SUBAPPLICATION mapping_Uebung_033_VV_FORTE_PC_B (* LED Strip Blinkende LED *)
  (* Standard: 61499-2 *)
  (* Version 1.0, 2023-10-23, franz *)
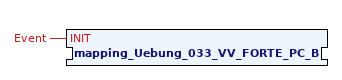
  EVENT_INPUT
    INIT;
  END_EVENT
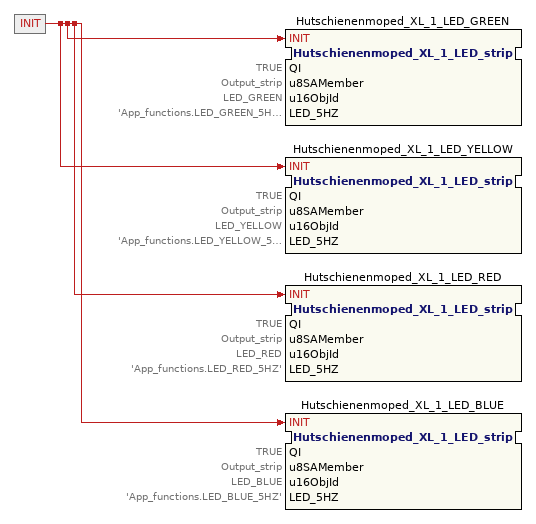
  FBS
    Hutschienenmoped_XL_1_LED_YELLOW : Hutschienenmoped_XL_1_LED_strip(QI := TRUE, u8SAMember := Output_strip, u16ObjId := LED_YELLOW, LED_5HZ := 'App_functions.LED_YELLOW_5HZ');
    Hutschienenmoped_XL_1_LED_GREEN : Hutschienenmoped_XL_1_LED_strip(QI := TRUE, u8SAMember := Output_strip, u16ObjId := LED_GREEN, LED_5HZ := 'App_functions.LED_GREEN_5HZ');
    Hutschienenmoped_XL_1_LED_RED : Hutschienenmoped_XL_1_LED_strip(QI := TRUE, u8SAMember := Output_strip, u16ObjId := LED_RED, LED_5HZ := 'App_functions.LED_RED_5HZ');
    Hutschienenmoped_XL_1_LED_BLUE : Hutschienenmoped_XL_1_LED_strip(QI := TRUE, u8SAMember := Output_strip, u16ObjId := LED_BLUE, LED_5HZ := 'App_functions.LED_BLUE_5HZ');
  END_FBS
  EVENT_CONNECTIONS
    INIT TO Hutschienenmoped_XL_1_LED_YELLOW.INIT;
    INIT TO Hutschienenmoped_XL_1_LED_GREEN.INIT;
    INIT TO Hutschienenmoped_XL_1_LED_RED.INIT;
    INIT TO Hutschienenmoped_XL_1_LED_BLUE.INIT;
  END_CONNECTIONS
END_SUBAPPLICATION
